(*
SPDX-FileCopyrightText: © 2026 Oleksandr Tiutyk <trofimich@gmail.com>
SPDX-License-Identifier: MIT
License: https://opensource.org/license/mit
*)

(*!
<summary>Initializes automation components and advances their cyclic execution.</summary>
<description>
FB_init borrows the root array. Its storage and components must outlive all runner calls. Keep its bounds,
slot identities and order fixed. Each root instance must occupy exactly one slot. The runner uses this binding from one task.
Execute updates system services, services the calling task's LogManager destination and processes components
according to the runner state. Its normal epilogue clears the exception payload and releases registered
auto-disposed objects. Call outside handlers that swallow fatal runtime exceptions.
</description>
*)

{attribute 'no_explicit_call' := 'do not call this function block directly'}
FUNCTION_BLOCK AutomationRunner EXTENDS TOF_Core.Object IMPLEMENTS IAutomationRunner
VAR_OUTPUT
	InitializationErrorMessage : TOF_Core.ERROR_MESSAGE;
END_VAR
VAR_STAT
	{attribute 'hide'} 
	_ClassName : STRING := __POUNAME();
END_VAR
VAR
	{attribute 'hide'} 
	_State : AUTOMATION_RUNNER_STATE;
	_Components : POINTER TO IAutomationComponent;
	_FirstIndex : DINT;
	_LastIndex : DINT;
	_RootsValidated : BOOL;
END_VAR

(*!
<summary>Gets the class name of the runner.</summary>
*)
{attribute 'monitoring' := 'call'}
PROPERTY ClassName : REFERENCE TO STRING
GET
ClassName REF= _ClassName;
END_GET
END_PROPERTY

(*!
<summary>Initializes or executes the constructor-bound roots in array order.</summary>
<description>
Once system data is ready, the runner checks the complete root array before initializing any root.
An empty array, null slot or repeated root makes the runner INVALID. Duplicate diagnostics identify both array indices.
Call from the outer task boundary. Nested runner execution is unsupported because cleanup covers the calling task.
Call outside recoverable handlers. Services the current task logger through LogManager.ExecuteCurrentTaskLogger on each call.
A registry allocation failure caught by a callback is raised again at FINAL_ACTIONS.
</description>
*)

METHOD FINAL Execute
VAR
	i : LINT;
	component : IAutomationComponent;
			
	initialized : BOOL;
END_VAR
TOF_Core.System.Execute();		

TOF_Core.LogManager.ExecuteCurrentTaskLogger();

IF TOF_Core.System.SystemDataValid THEN
	CASE _State OF
		AUTOMATION_RUNNER_STATE.INITIALIZING:
			IF NOT _RootsValidated THEN
				InitializationErrorMessage := getRootConfigurationError();

				IF InitializationErrorMessage <> "" THEN
					_State := AUTOMATION_RUNNER_STATE.INVALID;
					JMP FINAL_ACTIONS;
				END_IF

				_RootsValidated := TRUE;
			END_IF

			initialized := TRUE;
			
			FOR i := _FirstIndex TO _LastIndex DO
				component := _Components[TO_UDINT(i - _FirstIndex)];

				IF component = 0 THEN
					_State := AUTOMATION_RUNNER_STATE.INVALID;					
					InitializationErrorMessage := TOF_Core.WideStrings.Concat255("controller[", TO_WSTRING(i), "] is null");					
					JMP FINAL_ACTIONS;					
				END_IF

				component.Initialize();
				
				CASE component.OperationalState OF
					OPERATIONAL_STATE.INVALID:
						_State := AUTOMATION_RUNNER_STATE.INVALID;

						IF TOF_Core.WideStrings.IsNullOrWhiteSpace(stringToCheck := component.OperationalStateReason) THEN
							InitializationErrorMessage := TOF_Core.WideStrings.Concat255(
								"controller[",
								TO_WSTRING(i),
								"] (",
								component.Name,
								") failed"
							);
						ELSE
							InitializationErrorMessage := TOF_Core.WideStrings.Concat255(
								"controller[",
								TO_WSTRING(i),
								"] (",
								component.Name,
								") failed: ",
								component.OperationalStateReason
							);
						END_IF

						JMP FINAL_ACTIONS;
						
					OPERATIONAL_STATE.INITIALIZING:
						initialized := FALSE;						
				END_CASE
			END_FOR		
			
			IF initialized THEN
				_State := AUTOMATION_RUNNER_STATE.RUNNING;
			END_IF
		
		AUTOMATION_RUNNER_STATE.RUNNING:
			FOR i := _FirstIndex TO _LastIndex DO
				component := _Components[TO_UDINT(i - _FirstIndex)];

				IF component <> 0 THEN
					component.Execute();
				END_IF
			END_FOR		
	END_CASE
END_IF

FINAL_ACTIONS:

TOF_Core.DynamicMemoryManager.RaiseIfAllocationFailed();

TOF_Core.ExceptionManager.Cleanup();
TOF_Core.DynamicMemoryManager.CleanupMemory();
END_METHOD

(*!
<summary>Returns the first configuration error in the bound root array, or an empty message on success.</summary>
<description>
Compares interface identities in slot order without invoking root callbacks. Indices use the caller's declared bounds.
</description>
*)
METHOD PRIVATE getRootConfigurationError : WSTRING(255)
VAR
	i : LINT;
	previousIndex : LINT;
	component : IAutomationComponent;
END_VAR
IF _Components = 0 OR_ELSE _LastIndex < _FirstIndex THEN
	getRootConfigurationError := "No controllers to run";
	RETURN;
END_IF

FOR i := _FirstIndex TO _LastIndex DO
	component := _Components[TO_UDINT(i - _FirstIndex)];

	IF component = 0 THEN
		getRootConfigurationError := TOF_Core.WideStrings.Concat255("controller[", TO_WSTRING(i), "] is null");
		RETURN;
	END_IF

	FOR previousIndex := _FirstIndex TO i - 1 DO
		IF _Components[TO_UDINT(previousIndex - _FirstIndex)] = component THEN
			getRootConfigurationError := TOF_Core.WideStrings.Concat255(
				"controller[",
				TO_WSTRING(i),
				"] duplicates controller[",
				TO_WSTRING(previousIndex),
				"]"
			);
			RETURN;
		END_IF
	END_FOR
END_FOR
END_METHOD

(*!
<summary>Binds the runner to the caller's root array for its lifetime.</summary>
<description>
Borrows storage and records the declared index bounds. Root validation and callbacks begin in Execute.
The caller keeps the array and its ordered component references valid for every call.
</description>
<param name="components">Array of automation roots in execution order.</param>
*)
METHOD FB_init : BOOL
VAR_INPUT
	bInitRetains : BOOL; // TRUE: the retain variables are initialized (reset warm / reset cold)
	bInCopyCode : BOOL; // TRUE: the instance will be copied to the copy code afterward (online change)
END_VAR
VAR_IN_OUT CONSTANT
	components : ARRAY [*] OF IAutomationComponent;
END_VAR
_FirstIndex := LOWER_BOUND(components, 1);
_LastIndex := UPPER_BOUND(components, 1);

IF _FirstIndex <= _LastIndex THEN
	_Components := components;
END_IF
END_METHOD

(*!
<summary>Gets the namespace of the runner.</summary>
*)
{attribute 'monitoring' := 'call'}
PROPERTY NamespaceName : REFERENCE TO STRING
GET
NamespaceName REF= CurrentNamespace.Name;
END_GET
END_PROPERTY

(*!
<summary>Gets instance memory footprint in bytes.</summary>
*)
{attribute 'monitoring' := 'call'}
PROPERTY SelfSize : ULINT
GET
SelfSize := XSIZEOF(THIS^);
END_GET
END_PROPERTY

(*!
<summary>Gets current runner state.</summary>
*)
{attribute 'monitoring' := 'call'}
PROPERTY FINAL State : AUTOMATION_RUNNER_STATE
GET
State := _State;
END_GET
END_PROPERTY

(*!
<summary>Gets string representation of current runner state.</summary>
*)
{attribute 'monitoring' := 'call'}
PROPERTY StateName : STRING
GET
StateName := TO_STRING(_State);
END_GET
END_PROPERTY

END_FUNCTION_BLOCK

(* stored: Version 1.1.0.1
   POU AutomationRunner: Id {91ad6e09-e217-437d-b360-1103f460a0a5}, SpecialFunc None
   Property ClassName: Id {12ea2f4d-4597-416e-8305-e7d74fbf4c45}
   Get Get: Id {9841726e-851b-4678-a1b5-99c8a1cc58e0}
   Method Execute: Id {16952208-3067-4c16-b350-7fd85c7e6a7d}
   Method getRootConfigurationError: Id {86163466-39f9-478e-95d9-8afe8b683141}
   Method FB_init: Id {9dcb424f-eaa9-4a0f-923f-5afac333563a}
   Property NamespaceName: Id {d334c947-0a4c-4dfb-8401-47625a37779f}
   Get Get: Id {bed6e691-78c8-4572-bc37-6f5114bddb38}
   Property SelfSize: Id {15159a07-9ebc-498d-b2b1-558ebf3db84b}
   Get Get: Id {8ba632cf-a14d-49ee-bd64-3903af43dc94}
   Property State: Id {01547c3c-4426-4f09-bee4-07d5ec475004}
   Get Get: Id {4d2a4364-3afa-4b24-8a3f-64df284a4352}
   Property StateName: Id {06754117-469e-4960-a8f1-83200cc43cd1}
   Get Get: Id {ba601b6a-9ce0-457e-ac1f-5e869698dcb9} *)
